// TIA Portal project "Başlangıç Kesmesi Uygulaması V1" (V16)
// Vorlageprojekt für das Buch mit Zielsystem S7-1200

(* hardware
DEVICE "S7-1200-Station_1"  S7-1200 Station
   slot 0: "Baugruppenträger_0"  Rack  V1.0
   slot 1: "PLC_1"  CPU 1214C DC/DC/DC  6ES7 214-1AG40-0XB0  V4.4
*)

// ===== PLC "PLC_1"  CPU 1214C DC/DC/DC =====

VAR_GLOBAL   // PLC tag table "Standard-Variablentabelle"
   "Sistem_Start_Mem" AT %M10.0 : Bool;
   "Kenar_Darbesi" AT %M10.1 : Bool;
   "Kenar_Darbesi_1" AT %M20.0 : Bool;
   "Kenar_Darbesi_2" AT %M20.1 : Bool;
   "Ürün_Sayısı" AT %MW40 : Int;
   "Tag_1" AT %M30.0 : Bool;
END_VAR

VAR_GLOBAL   // PLC tag table "Tag table_1"
   "Start_But" AT %I0.0 : Bool;
   "Stop_But" AT %I0.1 : Bool;
   "Sensör_1" AT %I0.4 : Bool;
   "Sayıcı_Ekranı" AT %QW30 : Int;
   "Konveyör_1" AT %Q0.0 : Bool;
   "Konveyör_2" AT %Q0.1 : Bool;
   "Konveyör_3" AT %Q0.2 : Bool;
   "Konveyör_4" AT %Q0.3 : Bool;
   "Sensör_2" AT %I0.5 : Bool;
   "Uyarı_Lambası" AT %Q0.5 : Bool;
   "Sürücü_İleride_Sensörü" AT %I0.3 : Bool;
   "Sürücü_Geride_Sensörü" AT %I0.2 : Bool;
   "Sürücü" AT %Q0.4 : Bool;
END_VAR

// folder: System blocks/Program resources

DATA_BLOCK "Tımer_1"   // DB1
{ S7_Optimized_Access := 'TRUE' }
AUTHOR : Simatic
FAMILY : IEC
NAME : IEC_TMR
VERSION : 1.0
// stored: InstanceOfName IEC_TIMER
"IEC_TIMER"
BEGIN
END_DATA_BLOCK

// folder: (top level)

FUNCTION "MHJ-PLC-Lab-Function-S71200" : Void   // FC9000, SCL
{ S7_Optimized_Access := 'TRUE' }
VERSION : 0.1
   VAR_TEMP
      rdTimeReturn : Int;
      outputTime : DTL;
      SyncVal : Byte;
      forVal : Int;
      forVal_2 : Int;
      Value : Byte;
   END_VAR
   VAR CONSTANT
      CompVal : Byte := 16#34;
      Value_01 : Byte := 16#11;
      Value_01_DW : DWord := 16#A165_D992;
      Value_02_DW : DWord := 16#58BE_4401;
   END_VAR
BEGIN

   #Value:=PEEK(area := 16#82,
        dbNumber := 0,
        byteOffset := 511);
   #Value := #Value + 1;

   POKE(area := 16#82,
        dbNumber := 0,
        byteOffset := 511,
        value := #Value);

   POKE(area:=16#81,
        dbNumber:=0,
        byteOffset:=1016,
        value:=#Value_01_DW);
   POKE(area := 16#81,
        dbNumber := 0,
        byteOffset := 1020,
        value := #Value_02_DW);

   POKE(area := 16#81,
        dbNumber := 0,
        byteOffset := 511,
        value := B#16#00);

   FOR #forVal := 0 TO 120 DO
       FOR #forVal_2:=0 TO 10 DO
           #rdTimeReturn:=RD_SYS_T(#outputTime);
           #rdTimeReturn := WR_SYS_T(#outputTime);
           #rdTimeReturn := RD_SYS_T(#outputTime);
           #rdTimeReturn := WR_SYS_T(#outputTime);
       END_FOR;
       #SyncVal:= PEEK(area := 16#81,
                      dbNumber := 0,
                      byteOffset := 511);
       IF #SyncVal = #CompVal THEN
          GOTO M_1;
       END_IF;
   END_FOR;
   RETURN;

   M_1:
   POKE(area := 16#81,
        dbNumber := 0,
        byteOffset := 511,
        value := B#16#0);
END_FUNCTION

ORGANIZATION_BLOCK "Main"   // OB1, LAD, ProgramCycle
TITLE = "Main Program Sweep (Cycle)"
{ S7_Optimized_Access := 'TRUE' }
VERSION : 0.1
   VAR_INPUT
      Initial_Call : Bool;   // Initial call of this OB
      Remanence : Bool;   // =True, if remanent data are available
   END_VAR
   VAR_TEMP   // added for the SCL form of the ladder/FBD networks
      _w1 : Bool;
   END_VAR
BEGIN

REGION Network 1: Connection block for PLCSIM communications. Don't delete this network!
   // Im Netzwerk 1 wird der Konnektierungsbaustein für PLC-Lab aufgerufen.
   // Dieser Aufruf darf nicht entfernt werden!
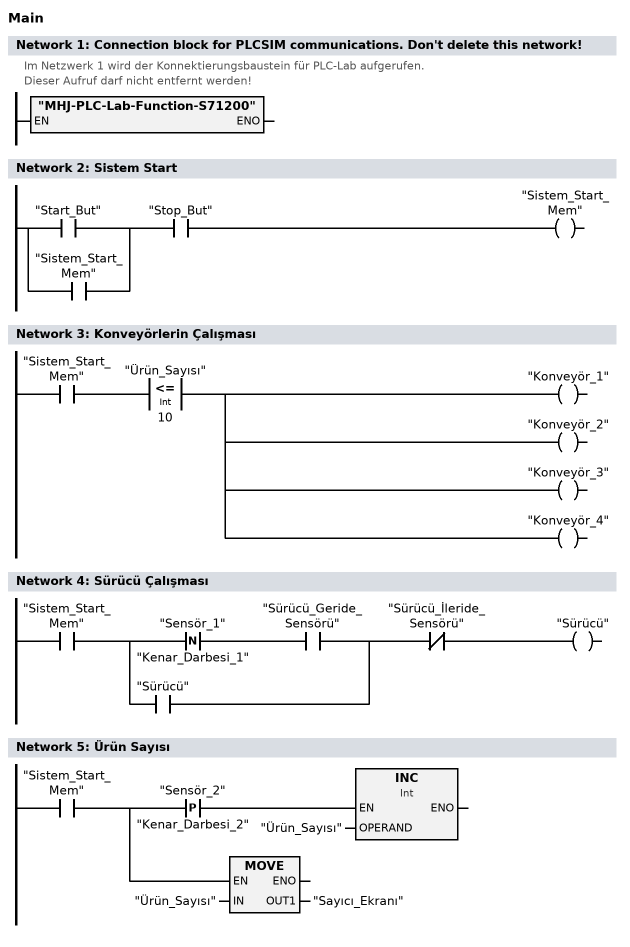
   RUNG wire#powerrail
      "MHJ-PLC-Lab-Function-S71200"()
   END_RUNG
   // the same network as SCL:
   "MHJ-PLC-Lab-Function-S71200"();
END_REGION

REGION Network 2: Sistem Start
   RUNG wire#powerrail
      Contact( "Start_But" )
      wire#w1
      Contact( "Stop_But" )
      Coil( "Sistem_Start_Mem" )
   END_RUNG
   RUNG wire#powerrail
      Contact( "Sistem_Start_Mem" )
   END_RUNG wire#w1
   // the same network as SCL:
   "Sistem_Start_Mem" := ("Start_But" OR "Sistem_Start_Mem") AND "Stop_But";
END_REGION

REGION Network 3: Konveyörlerin Çalışması
   RUNG wire#powerrail
      Contact( "Sistem_Start_Mem" )
      { S7_Templates := "SrcType := Int" } LE_Contact(in1 := "Ürün_Sayısı", in2 := 10)
      wire#w1
      Coil( "Konveyör_1" )
   END_RUNG
   RUNG wire#w1
      Coil( "Konveyör_2" )
   END_RUNG
   RUNG wire#w1
      Coil( "Konveyör_3" )
   END_RUNG
   RUNG wire#w1
      Coil( "Konveyör_4" )
   END_RUNG
   // the same network as SCL:
   "Konveyör_1" := "Sistem_Start_Mem" AND ("Ürün_Sayısı" <= 10);
   "Konveyör_2" := "Konveyör_1";
   "Konveyör_3" := "Konveyör_1";
   "Konveyör_4" := "Konveyör_1";
END_REGION

REGION Network 4: Sürücü Çalışması
   RUNG wire#powerrail
      Contact( "Sistem_Start_Mem" )
      wire#w1
      N_Contact(operand := "Sensör_1", bit := "Kenar_Darbesi_1")
      Contact( "Sürücü_Geride_Sensörü" )
      wire#w2
      I_Contact( "Sürücü_İleride_Sensörü" )
      Coil( "Sürücü" )
   END_RUNG
   RUNG wire#w1
      Contact( "Sürücü" )
   END_RUNG wire#w2
   // the same network as SCL:
   #_w1 := "Sistem_Start_Mem" AND NOT "Sensör_1" AND "Kenar_Darbesi_1";   // falling edge of "Sensör_1"
   "Kenar_Darbesi_1" := "Sensör_1";
   "Sürücü" := ((#_w1 AND "Sürücü_Geride_Sensörü") OR ("Sistem_Start_Mem" AND "Sürücü")) AND NOT "Sürücü_İleride_Sensörü";
END_REGION

REGION Network 5: Ürün Sayısı
   RUNG wire#powerrail
      Contact( "Sistem_Start_Mem" )
      wire#w1
      P_Contact(operand := "Sensör_2", bit := "Kenar_Darbesi_2")
      { S7_Templates := "DestType := Int" } Inc( "Ürün_Sayısı" )
   END_RUNG
   RUNG wire#w1
      Move(in := "Ürün_Sayısı", out1 => "Sayıcı_Ekranı")
   END_RUNG
   // the same network as SCL:
   #_w1 := "Sistem_Start_Mem" AND "Sensör_2" AND NOT "Kenar_Darbesi_2";   // rising edge of "Sensör_2"
   "Kenar_Darbesi_2" := "Sensör_2";
   IF #_w1 THEN "Ürün_Sayısı" := "Ürün_Sayısı" + 1; END_IF;
   IF "Sistem_Start_Mem" THEN "Sayıcı_Ekranı" := "Ürün_Sayısı"; END_IF;
END_REGION
END_ORGANIZATION_BLOCK

ORGANIZATION_BLOCK "Startup"   // OB100, LAD, Startup
TITLE = "Complete Restart"
{ S7_Optimized_Access := 'TRUE' }
VERSION : 0.1
   VAR_INPUT
      LostRetentive : Bool;   // True if retentive data are lost
      LostRTC : Bool;   // True if date and time are lost
   END_VAR
BEGIN

REGION Network 1: Çalışma Süresi
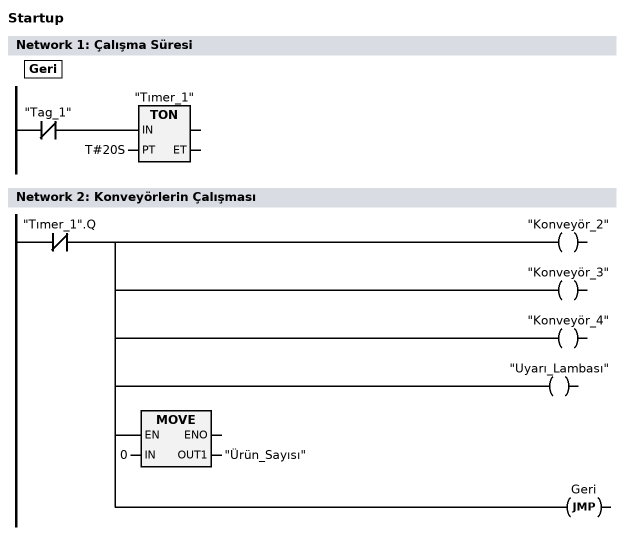
   Geri:
   "Tımer_1".TON(IN := NOT "Tag_1", PT := T#20S);
END_REGION

REGION Network 2: Konveyörlerin Çalışması
   RUNG wire#powerrail
      I_Contact( "Tımer_1".Q )
      wire#w1
      Coil( "Konveyör_2" )
   END_RUNG
   RUNG wire#w1
      Coil( "Konveyör_3" )
   END_RUNG
   RUNG wire#w1
      Coil( "Konveyör_4" )
   END_RUNG
   RUNG wire#w1
      Coil( "Uyarı_Lambası" )
   END_RUNG
   RUNG wire#w1
      Move(in := 0, out1 => "Ürün_Sayısı")
   END_RUNG
   RUNG wire#w1
      JumpCoil( Geri )
   END_RUNG
   // the same network as SCL:
   "Konveyör_2" := NOT "Tımer_1".Q;
   "Konveyör_3" := NOT "Tımer_1".Q;
   "Konveyör_4" := NOT "Tımer_1".Q;
   "Uyarı_Lambası" := NOT "Tımer_1".Q;
   IF NOT "Tımer_1".Q THEN
       "Ürün_Sayısı" := 0;
       GOTO Geri;
   END_IF;
END_REGION
END_ORGANIZATION_BLOCK